FUNCTION_BLOCK IVController
VAR
    inputRequest1  AT %Q* : ProcessData1;
    inputResponse1 AT %I* : ProcessData1;
    statusOfSystem AT %I* : StatusCam;
    _trigger              : BOOL;
    _readString           : BOOL;
    _readDeviceInfo       : BOOL;
END_VAR
VAR
    InfoData AT %I* : InfoData;
    WcState  AT %I* : WcState;
END_VAR

VAR
    _fb_coe_write       : FB_EcCoESdoWrite; // Function Block for writing in CoE
    _fb_coe_read        : FB_EcCoESdoRead;  // Function Block for reading from CoE
    userNetId           : T_AmsNetId;       // Have to be entered
    _startWrite         : BOOL := FALSE;    // Sign for start writing
    _startRead          : BOOL := FALSE;    // Sign for start reading
    _nState             : BYTE := 0;        // RW-status
    _int16Buffer        : INT;              // Buffer for reading
    _uint16Buffer       : UINT := 22;       // Buffer for writing
    _bTxPDOState AT %I* : BOOL;             // (PDO for synchronization)
    AdsErrId            : UDINT;
    CANopenErrId        : UDINT;

    _index             : UINT := 16#1008;
    _subIndex          : BYTE := 0;
    _result            : STRING;
    _stringBuffer      : STRING;
    _numberBuffer      : UDINT;
    _exe               : BOOL;
    _generalDeviceInfo : GeneralDeviceInformation;
    _IdentityCoe       : IdentityCoe;
    _coordinates       : Coordinates;
    _readCoordinates   : BOOL;
END_VAR

IF _trigger THEN
    inputRequest1.stProcessData.Trigger := TRUE;

    IF inputResponse1.stProcessData.Trigger THEN
        _trigger                            := FALSE;
        inputRequest1.stProcessData.Trigger := FALSE;
    end_if
END_IF

userNetId := Tc2_System.F_CreateAmsNetId(infodata.AdsAddr.netId);

IF _readString THEN
    _stringBuffer := CoeReadString(_index := _index, _subIndex := _subIndex);
END_IF

IF _readDeviceInfo THEN

    IF GeneralDeviceInfo() THEN
        _readDeviceInfo := false;
    END_IF
END_IF

CoeReadIdentity();

IF _readCoordinates THEN
    IF CoeReadCoordinates() THEN
        _readCoordinates := FALSE;
    END_IF

END_IF

METHOD CoeReadCoordinates : BOOL
VAR_INST
    step : UINT := 1;

END_VAR
CASE step OF
    1:
        CoeReadCoordinates := FALSE;
        step               := 10;
    10:
        _coordinates.xValue := CoeReadUDINT
        (
            _index      := 16#8015
            , _subIndex := 16#11
        );

        IF NOT _fb_coe_read.bBusy THEN
            step := 20;
        END_IF
    20:
        _coordinates.yValue := CoeReadUDINT
        (
            _index      := 16#8015
            , _subIndex := 16#12
        );

        IF NOT _fb_coe_read.bBusy THEN
            step := 40;
        END_IF
    40:
        _coordinates.angleValue := CoeReadUDINT
        (
            _index      := 16#8015
            , _subIndex := 16#13
        );

        IF NOT _fb_coe_read.bBusy THEN
            step               := 1;
            CoeReadCoordinates := TRUE;
        END_IF
END_CASE
END_METHOD

METHOD CoeReadIdentity : UDINT
VAR_INST
    _fb_coe_read_ext   : Tc2_EtherCAT.FB_EcCoESdoReadEx;
    _timeout           : TIME := DEFAULT_ADS_TIMEOUT;
    _identityCoeToSwap : IdentityCoe;

    i     : UINT;
    _test : STRING;
END_VAR

// Read entry
_fb_coe_read_ext
(
    sNetId            := userNetId
    , nSlaveAddr      := InfoData.AdsAddr.port
    , nSubIndex       := 0
    , nIndex          := 16#1018
    , pDstBuf         := ADR(_identityCoeToSwap)
    , cbBufLen        := 32
    , bExecute        := true
    , tTimeout        := _timeout
    , bCompleteAccess := TRUE
);

IF _fb_coe_read.bError THEN
    _nState := 100; // Error case
ELSE

    IF NOT _fb_coe_read.bBusy THEN
        _IdentityCoe.ProductKey   := SHR(_identityCoeToSwap.ProductKey, 16);
        _IdentityCoe.VendorId     := SHR(_identityCoeToSwap.VendorId, 16);
        _IdentityCoe.Revision     := SHR(_identityCoeToSwap.Revision, 16);
        _IdentityCoe.SerialNumber := SHR(_identityCoeToSwap.SerialNumber, 16);
        _fb_coe_read(bExecute := FALSE);
        _readString := false;
    END_IF

END_IF
END_METHOD

METHOD CoeReadString : STRING
//VAR_INST
//    _stringBuffer : STRING;
//END_VAR
VAR_INPUT
    _index    : UINT;
    _subIndex : BYTE;
END_VAR

// Read entry
_fb_coe_read
(
    sNetId       := userNetId
    , nSlaveAddr := InfoData.AdsAddr.port
    //    , nSlaveAddr := 1001
    , nSubIndex := _subIndex
    , nIndex    := _index
    , pDstBuf   := ADR(_stringBuffer)
    , cbBufLen  := 12
    , bExecute  := true
    , tTimeout  := T#1S
);

IF _fb_coe_read.bError THEN
    AdsErrId := _fb_coe_read.nErrId;
ELSE
    IF NOT _fb_coe_read.bBusy THEN
        _fb_coe_read(bExecute := FALSE);
        _readString := false;
    END_IF
END_IF

CoeReadString := _stringBuffer;
END_METHOD

METHOD CoeReadUDINT : UDINT
//VAR_INST
//    _stringBuffer : STRING;
//END_VAR
VAR_INPUT
    _index    : UINT;
    _subIndex : BYTE;
END_VAR

// Read entry
_fb_coe_read
(
    sNetId       := userNetId
    , nSlaveAddr := InfoData.AdsAddr.port
    //    , nSlaveAddr := 1001
    , nSubIndex := _subIndex
    , nIndex    := _index
    , pDstBuf   := ADR(_numberBuffer)
    , cbBufLen  := 32
    , bExecute  := true
    , tTimeout  := T#1S
);

IF _fb_coe_read.bError THEN
    _nState := 100; // Error case
ELSE
    IF NOT _fb_coe_read.bBusy THEN
        _fb_coe_read(bExecute := FALSE);
        _readString := false;
    END_IF
END_IF

CoeReadUDINT := _numberBuffer;
END_METHOD

METHOD PRIVATE GeneralDeviceInfo : BOOL;
VAR_INST
    step : UINT := 1;

END_VAR
CASE step OF
    1:
        GeneralDeviceInfo := FALSE;
        step              := 10;
    10:
        _generalDeviceInfo.DeviceName := CoeReadString
        (
            _index      := 16#1008
            , _subIndex := 0
        );

        IF NOT _fb_coe_read.bBusy THEN
            step := 20;
        END_IF
    20:
        step := 25;
    25:
        _generalDeviceInfo.HardwareVersion := CoeReadString
        (
            _index      := 16#1009
            , _subIndex := 0
        );

        IF NOT _fb_coe_read.bBusy THEN
            step := 30;
        END_IF
    30:
        step := 35;
    35:
        _generalDeviceInfo.DeviceType := CoeReadUDINT
        (
            _index      := 16#1000
            , _subIndex := 0
        );

        IF NOT _fb_coe_read.bBusy THEN
            step := 40;
        END_IF
    40:
        GeneralDeviceInfo := FALSE;
        step              := 45;
    45:
        _generalDeviceInfo.SoftwareVersion := CoeReadString
        (
            _index      := 16#100A
            , _subIndex := 0
        );

        IF NOT _fb_coe_read.bBusy THEN
            step              := 1;
            GeneralDeviceInfo := TRUE;
        END_IF

END_CASE
END_METHOD

END_FUNCTION_BLOCK

(* stored: Version 1.1.0.1, ProductVersion 3.1.4024.12
   POU IVController: Id {fe008e94-684c-4663-a099-492675947df8}, SpecialFunc None
   Folder CoeActions: Id {1a3a42f9-6ee0-40e3-b164-d0a1d9218ddf}
   Method CoeReadCoordinates: Id {f40c82fa-d496-4376-832a-992a794686e2}
   Method CoeReadIdentity: Id {c7eb3a96-f07b-4390-8e80-9ae055189873}
   Method CoeReadString: Id {606533e4-95ef-4d2f-875f-216f57b356b2}
   Method CoeReadUDINT: Id {b0ff3618-3656-4acd-9fa0-c2d775da4f39}
   Method GeneralDeviceInfo: Id {71ed06fb-4056-430e-b650-3eb8d00d0129} *)
